// TIA Portal V18 export
ORGANIZATION_BLOCK "Main"   // OB1, LAD, ProgramCycle
TITLE = "Main Program Sweep (Cycle)"
{ S7_Optimized_Access := 'TRUE' }
VERSION : 0.1
// stored: AutoNumber true, IsIECCheckEnabled true, SetENOAutomatically false
   VAR_INPUT
      Initial_Call : Bool;   // Initial call of this OB
      Remanence : Bool;   // =True, if remanent data are available
   END_VAR
BEGIN

REGION Network 1: call conveyor
   // //=============================================================================
   // //Siemens AG // (c)Copyright (2018)
   // //-----------------------------------------------------------------------------
   // // Library: (that the source is dedicated to)
   // // Tested with: (test system with FW version)
   // // Engineering: TIA Portal V15
   // // Restrictions: (OB types, etc.)
   // // Requirements: (hardware, technological package, memory needed, etc.)
   // // Functionality: (that is implemented in the block)
   // //-----------------------------------------------------------------------------
   // // Change log table:
   // // Version Date Expert in charge Changes applied
   // // 24.08.18 dd.mm.yyyy (Name of expert) First released version
   // //=============================================================================
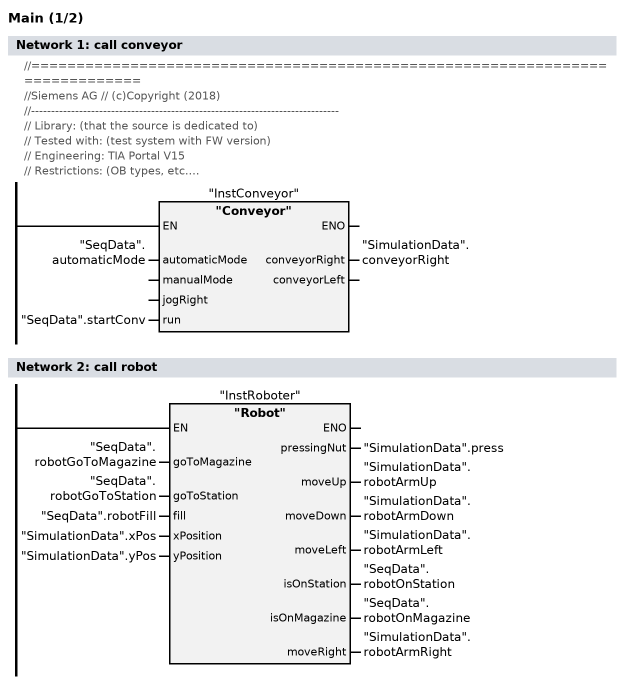
   RUNG wire#powerrail
      "InstConveyor"(automaticMode := "SeqData".automaticMode, manualMode :=, jogRight :=, run := "SeqData".startConv, conveyorRight => "SimulationData".conveyorRight, conveyorLeft =>)
   END_RUNG
   // the same network as SCL:
   "InstConveyor"(automaticMode := "SeqData".automaticMode,   // "Conveyor"
                  run := "SeqData".startConv,
                  conveyorRight => "SimulationData".conveyorRight);
END_REGION

REGION Network 2: call robot
   RUNG wire#powerrail
      "InstRoboter"(goToMagazine := "SeqData".robotGoToMagazine, goToStation := "SeqData".robotGoToStation, fill := "SeqData".robotFill, xPosition := "SimulationData".xPos, yPosition := "SimulationData".yPos, pressingNut => "SimulationData".press, moveUp => "SimulationData".robotArmUp, moveDown => "SimulationData".robotArmDown, moveLeft => "SimulationData".robotArmLeft, isOnStation => "SeqData".robotOnStation, isOnMagazine => "SeqData".robotOnMagazine, moveRight => "SimulationData".robotArmRight)
   END_RUNG
   // the same network as SCL:
   "InstRoboter"(goToMagazine := "SeqData".robotGoToMagazine,   // "Robot"
                 goToStation := "SeqData".robotGoToStation,
                 fill := "SeqData".robotFill,
                 xPosition := "SimulationData".xPos,
                 yPosition := "SimulationData".yPos,
                 pressingNut => "SimulationData".press,
                 moveUp => "SimulationData".robotArmUp,
                 moveDown => "SimulationData".robotArmDown,
                 moveLeft => "SimulationData".robotArmLeft,
                 isOnStation => "SeqData".robotOnStation,
                 isOnMagazine => "SeqData".robotOnMagazine,
                 moveRight => "SimulationData".robotArmRight);
END_REGION

REGION Network 3: call sequencer
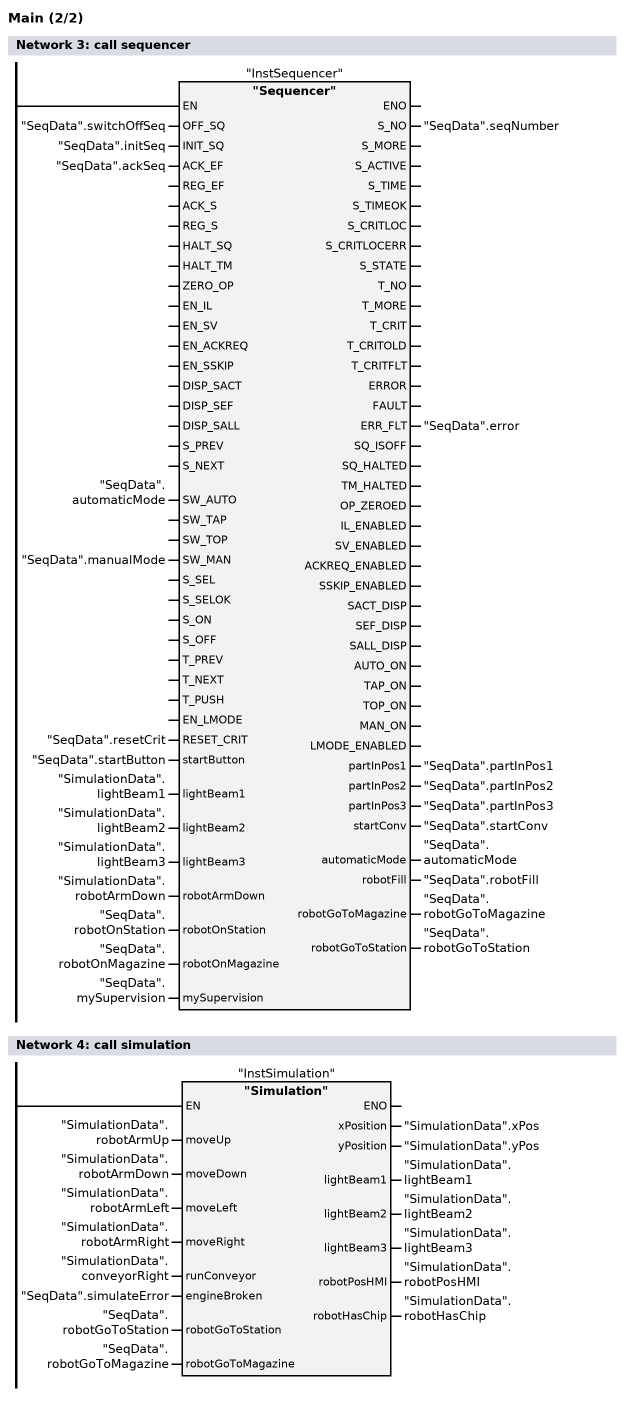
   RUNG wire#powerrail
      "InstSequencer"(OFF_SQ := "SeqData".switchOffSeq, INIT_SQ := "SeqData".initSeq, ACK_EF := "SeqData".ackSeq, REG_EF :=, ACK_S :=, REG_S :=, HALT_SQ :=, HALT_TM :=, ZERO_OP :=, EN_IL :=, EN_SV :=, EN_ACKREQ :=, EN_SSKIP :=, DISP_SACT :=, DISP_SEF :=, DISP_SALL :=, S_PREV :=, S_NEXT :=, SW_AUTO := "SeqData".automaticMode, SW_TAP :=, SW_TOP :=, SW_MAN := "SeqData".manualMode, S_SEL :=, S_SELOK :=, S_ON :=, S_OFF :=, T_PREV :=, T_NEXT :=, T_PUSH :=, EN_LMODE :=, RESET_CRIT := "SeqData".resetCrit, startButton := "SeqData".startButton, lightBeam1 := "SimulationData".lightBeam1, lightBeam2 := "SimulationData".lightBeam2, lightBeam3 := "SimulationData".lightBeam3, robotArmDown := "SimulationData".robotArmDown, robotOnStation := "SeqData".robotOnStation, robotOnMagazine := "SeqData".robotOnMagazine, mySupervision := "SeqData".mySupervision, S_NO => "SeqData".seqNumber, S_MORE =>, S_ACTIVE =>, S_TIME =>, S_TIMEOK =>, S_CRITLOC =>, S_CRITLOCERR =>, S_STATE =>, T_NO =>, T_MORE =>, T_CRIT =>, T_CRITOLD =>, T_CRITFLT =>, ERROR =>, FAULT =>, ERR_FLT => "SeqData".error, SQ_ISOFF =>, SQ_HALTED =>, TM_HALTED =>, OP_ZEROED =>, IL_ENABLED =>, SV_ENABLED =>, ACKREQ_ENABLED =>, SSKIP_ENABLED =>, SACT_DISP =>, SEF_DISP =>, SALL_DISP =>, AUTO_ON =>, TAP_ON =>, TOP_ON =>, MAN_ON =>, LMODE_ENABLED =>, partInPos1 => "SeqData".partInPos1, partInPos2 => "SeqData".partInPos2, partInPos3 => "SeqData".partInPos3, startConv => "SeqData".startConv, automaticMode => "SeqData".automaticMode, robotFill => "SeqData".robotFill, robotGoToMagazine => "SeqData".robotGoToMagazine, robotGoToStation => "SeqData".robotGoToStation)
   END_RUNG
   // the same network as SCL:
   "InstSequencer"(OFF_SQ := "SeqData".switchOffSeq,   // "Sequencer"
                   INIT_SQ := "SeqData".initSeq,
                   ACK_EF := "SeqData".ackSeq,
                   SW_AUTO := "SeqData".automaticMode,
                   SW_MAN := "SeqData".manualMode,
                   RESET_CRIT := "SeqData".resetCrit,
                   startButton := "SeqData".startButton,
                   lightBeam1 := "SimulationData".lightBeam1,
                   lightBeam2 := "SimulationData".lightBeam2,
                   lightBeam3 := "SimulationData".lightBeam3,
                   robotArmDown := "SimulationData".robotArmDown,
                   robotOnStation := "SeqData".robotOnStation,
                   robotOnMagazine := "SeqData".robotOnMagazine,
                   mySupervision := "SeqData".mySupervision,
                   S_NO => "SeqData".seqNumber,
                   ERR_FLT => "SeqData".error,
                   partInPos1 => "SeqData".partInPos1,
                   partInPos2 => "SeqData".partInPos2,
                   partInPos3 => "SeqData".partInPos3,
                   startConv => "SeqData".startConv,
                   automaticMode => "SeqData".automaticMode,
                   robotFill => "SeqData".robotFill,
                   robotGoToMagazine => "SeqData".robotGoToMagazine,
                   robotGoToStation => "SeqData".robotGoToStation);
END_REGION

REGION Network 4: call simulation
   RUNG wire#powerrail
      "InstSimulation"(moveUp := "SimulationData".robotArmUp, moveDown := "SimulationData".robotArmDown, moveLeft := "SimulationData".robotArmLeft, moveRight := "SimulationData".robotArmRight, runConveyor := "SimulationData".conveyorRight, engineBroken := "SeqData".simulateError, robotGoToStation := "SeqData".robotGoToStation, robotGoToMagazine := "SeqData".robotGoToMagazine, xPosition => "SimulationData".xPos, yPosition => "SimulationData".yPos, lightBeam1 => "SimulationData".lightBeam1, lightBeam2 => "SimulationData".lightBeam2, lightBeam3 => "SimulationData".lightBeam3, robotPosHMI => "SimulationData".robotPosHMI, robotHasChip => "SimulationData".robotHasChip)
   END_RUNG
   // the same network as SCL:
   "InstSimulation"(moveUp := "SimulationData".robotArmUp,   // "Simulation"
                    moveDown := "SimulationData".robotArmDown,
                    moveLeft := "SimulationData".robotArmLeft,
                    moveRight := "SimulationData".robotArmRight,
                    runConveyor := "SimulationData".conveyorRight,
                    engineBroken := "SeqData".simulateError,
                    robotGoToStation := "SeqData".robotGoToStation,
                    robotGoToMagazine := "SeqData".robotGoToMagazine,
                    xPosition => "SimulationData".xPos,
                    yPosition => "SimulationData".yPos,
                    lightBeam1 => "SimulationData".lightBeam1,
                    lightBeam2 => "SimulationData".lightBeam2,
                    lightBeam3 => "SimulationData".lightBeam3,
                    robotPosHMI => "SimulationData".robotPosHMI,
                    robotHasChip => "SimulationData".robotHasChip);
END_REGION
END_ORGANIZATION_BLOCK
